FUNCTION CACOS : complex
VAR_INPUT
	X : complex;
END_VAR
VAR
	Y : complex;
END_VAR

(*
version 1.0	21 feb 2008
programmer 	hugo
tested by	oscat

this function calculates the arcus cosinus function of a complex number

*)

y := CACOSH(x);
CACOS.re := y.im;
CACOS.im := -y.re;



(* revision history
hm	21. feb 2008	rev 1.0
	original version


*)

END_FUNCTION

(* stored: Version 1.1.0.1, ProductVersion 3.1.4024.9
   POU CACOS: Id {a7536260-5b3f-4ec3-a6ec-1077de90e06c}, SpecialFunc None *)
